TYPE "ADP.Decoded.Flash.UDT"
VERSION : 0.1
   STRUCT
      off : String[8] := 'off';
      on : String[8] := 'on';
   END_STRUCT;

END_TYPE

